# EPICS substitutions: knr1050Sup/knr1050_errors.substitutions
## Errors are not forwarded in protocol redirects
file "$(UTILITIES)/db/error_setter.template" {
  pattern {P, STREAM_PV, PV_NAME}
    {"\$(P)", "PRESSURE:LIMITS", "PRESSURE:MIN"}
    {"\$(P)", "PRESSURE:LIMITS", "PRESSURE:MAX"}
}
